FUNCTION_BLOCK QX_Emulated (* Composite FB wrapping other FBs *)
  (* Standard: 61499-2 *)
  (* Version 1.0, 2021-08-05, dorofeev *)
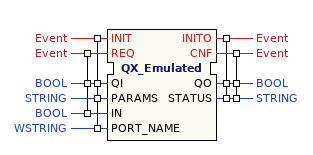
  EVENT_INPUT
    INIT WITH PORT_NAME, PARAMS, QI; (* Initialization Request *)
    REQ WITH IN, QI; (* Normal Execution Request *)
  END_EVENT
  EVENT_OUTPUT
    INITO WITH STATUS, QO; (* Initialization Confirm *)
    CNF WITH STATUS, QO; (* Execution Confirmation *)
  END_EVENT
  VAR_INPUT
    QI : BOOL; (* Input event qualifier *)
    PARAMS : STRING;
    IN : BOOL;
    PORT_NAME : WSTRING;
  END_VAR
  VAR_OUTPUT
    QO : BOOL; (* Output event qualifier *)
    STATUS : STRING;
  END_VAR
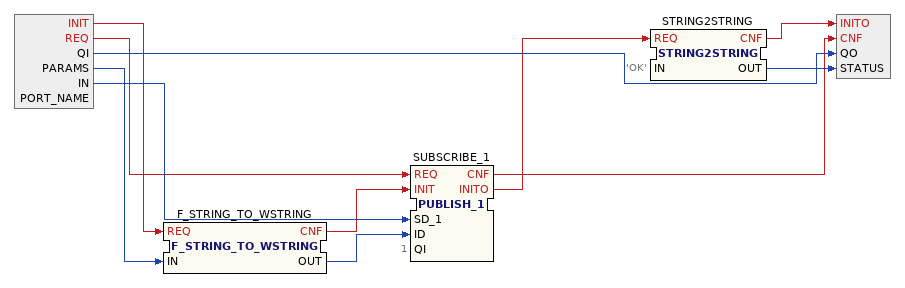
  FBS
    STRING2STRING : STRING2STRING(IN := 'OK');
    SUBSCRIBE_1 : PUBLISH_1(QI := 1);
    F_STRING_TO_WSTRING : F_STRING_TO_WSTRING;
  END_FBS
  EVENT_CONNECTIONS
    STRING2STRING.CNF TO INITO;
    SUBSCRIBE_1.CNF TO CNF;
    SUBSCRIBE_1.INITO TO STRING2STRING.REQ;
    REQ TO SUBSCRIBE_1.REQ;
    F_STRING_TO_WSTRING.CNF TO SUBSCRIBE_1.INIT;
    INIT TO F_STRING_TO_WSTRING.REQ;
  END_CONNECTIONS
  DATA_CONNECTIONS
    QI TO QO;
    STRING2STRING.OUT TO STATUS;
    IN TO SUBSCRIBE_1.SD_1;
    F_STRING_TO_WSTRING.OUT TO SUBSCRIBE_1.ID;
    PARAMS TO F_STRING_TO_WSTRING.IN;
  END_CONNECTIONS
END_FUNCTION_BLOCK
